FUNCTION_BLOCK FB_SingleTankSV1Ext EXTENDS FB_SingleTankSV1
VAR
	sNameTask : STRING;
	bBusyTask : BOOL;
END_VAR

SUPER^();

PROPERTY BusyTask : BOOL
GET
BusyTask := bBusyTask;
END_GET
END_PROPERTY

METHOD RegisterTask : BOOL
VAR_INPUT
	sTask : STRING;
END_VAR
IF NOT bBusyTask THEN
	sNameTask := sTask;
	bBusyTask := true;
	RegisterTask := TRUE;
ELSE
	RegisterTask := FALSE;
END_IF
END_METHOD

PROPERTY TaskRegistered : string
GET
TaskRegistered := sNameTask;
END_GET
END_PROPERTY

METHOD UnRegisterTask : BOOL
VAR_INPUT
END_VAR
bBusyTask := FALSE;
sNameTask := '';
UnRegisterTask := true;
END_METHOD

END_FUNCTION_BLOCK

(* stored: Version 1.1.0.1, ProductVersion 3.1.4024.12
   POU FB_SingleTankSV1Ext: Id {bb81fd6c-115b-43ef-86f2-3e70850eaa40}, SpecialFunc None
   Property BusyTask: Id {5f01a18e-053c-4c41-b9ca-6269647a9d05}
   Get Get: Id {9ddb7b43-f3c9-4b96-a236-c8af6c9b47dc}
   Method RegisterTask: Id {b2b1d959-671e-4ae2-84ea-d47fee3ebd97}
   Property TaskRegistered: Id {61920fe3-7ea6-407c-8170-b26e9f608c7b}
   Get Get: Id {c1d10f15-aa36-451e-a62e-0ee8dc217b47}
   Method UnRegisterTask: Id {1e29d8d5-b2d1-4f66-8dea-ddba1177c4a3} *)
